(* CoDeSys 2.3 export: PACKML_STATEMODEL_20191003.EXP *)

(* Data type *)
TYPE E_Mode :
(*UserModes: Modes for different production states*)
(
	eMode_undefined := 0,
	eMode_Automatic :=1,
	eMode_Manual :=3,
	eMode_Production1 :=5,
	eMode_Production2 :=6
);
END_TYPE

(* Data type *)
TYPE E_ModeProc :
(*Procedural control modes. Can be changed in any state*)
(
	eModeProc_undefined := 0,
	eModeProc_Automatic :=1,
	eModeProc_SemiAutomatic :=2,
	eModeProc_Manual :=3
);
END_TYPE

(* Data type *)
TYPE E_PackMLState :
(*PackML States*)
(
	eSt_Aborting :=0,
	eSt_Aborted,
	eSt_Clearing,
	eSt_Stopped,
	eSt_Stopping,
	eSt_Resetting,
	eSt_Idle,
	eSt_Starting,
	eSt_Execute,
	eSt_Suspending,
	eSt_Suspended,
	eSt_Unsuspending,
	eSt_Holding,
	eSt_Held,
	eSt_UnHolding,
	eSt_Completing,
	eSt_Completed
);
END_TYPE

(* POU Examples/PRG_MAIN_SAMPLE, ST *)
PROGRAM PRG_MAIN_SAMPLE
VAR
(*	fbStateModel		: FB_PackMLStateModel_ST;	(*FB for executing PackML state model*)		*)
	bBlink				: BOOL;	(*1s blinkg for CodeSys Simulation*)
	c					: INT;	(*Support variable for blinking*)
END_VAR
(* ****** Section 1: Initialisations and default values. Initial conditions for variables on every PLC cycle*)
fbStateModel.bSC := FALSE;

(* ****** Section 2: Grouping PackML states for calling Programs or FB instances.
This is to avoid repetition inside case structure in Section 4. With IF clause setting lower (and upper) state limits we can filter out the states when we 
want to call specific programs. The order of states is defined in Tab:Data types > E_PackMLState. eSt_Aborting is the lowest and eSt_Completed is 
the highest. Here we filter out calling of the programs - we call them only when we are in higher states than Stopped. Inside IF there is again CASE 
which process each Control Mode separately.*)
(*Execution part. Making calls for program if we are on states above Stopped*)
IF (fbStateModel.eState > eSt_Stopped) THEN
	CASE fbStateModel.eMode OF
		(*MODE: MANUAL*)
		eMode_Manual:
			;
		(*MODE: AUTOMATIC*)
		eMode_Automatic:
			;
	END_CASE;
END_IF;

(* ****** Section 3: Actions in your program without considering the Control Mode. I.e. actions are performed same way indenpendent on
current Control Mode selection.*)
(*Mode independent state actions*)
CASE fbStateModel.eState OF
eSt_Aborting:
	(* One can make specific actions in case of specific Mode-State combination.
	   One can also consider to call a specific program when in specific Mode-State combination*)
	actAborting;
	fbStateModel.bSC := TRUE;		(*TODO: Remove/Replace this row with desired actions*)
eSt_Clearing:
	fbStateModel.bSC := TRUE;		(*TODO: Remove/Replace this row with desired actions*)
eSt_Stopping:
	fbStateModel.bSC := TRUE;		(*TODO: Remove/Replace this row with desired actions*)
eSt_Resetting:
	fbStateModel.bSC := TRUE;		(*TODO: Remove/Replace this row with desired actions*)
eSt_Holding:
	fbStateModel.bSC := TRUE;		(*TODO: Remove/Replace this row with desired actions*)
eSt_UnHolding:
	fbStateModel.bSC := TRUE;		(*TODO: Remove/Replace this row with desired actions*)
eSt_Suspending:
	fbStateModel.bSC := TRUE;		(*TODO: Remove/Replace this row with desired actions*)
eSt_Unsuspending:
	fbStateModel.bSC := TRUE;		(*TODO: Remove/Replace this row with desired actions*)
END_CASE;

(* ****** Section 4: Actions in your program which are Control Mode specific. Two nested case structures where outer one selects the
control mode and inner the PackML state. In order to avoid conflicts, it would be better to process each PackML state either in Section 3 
or Section 4, but not in both. *)
(*Execution mode related state actions*)
CASE fbStateModel.eMode OF
(*MODE: MANUAL*)
eMode_Manual:
	(* ****** Section 4.1: PackML state based processing actions when Control Mode is Manual.*)
	CASE fbStateModel.eState OF
	eSt_Idle:
		fbStateModel.bAck_Completed := FALSE;		(*TODO: Remove/Replace this row with desired actions*)
	eSt_Starting:
		fbStateModel.bSC := TRUE;					(*TODO: Remove/Replace this row with desired actions*)
	eSt_Completing:
		fbStateModel.bSC := TRUE;					(*TODO: Remove/Replace this row with desired actions*)
	eSt_Completed:
		fbStateModel.bAck_Completed := TRUE;		(*TODO: Remove/Replace this row with desired actions*)
	END_CASE;

(*MODE: AUTOMATIC*)
eMode_Automatic:
	(* ****** Section 4.2: PackML state based processing actions when Control Mode is Automatic.*)
	CASE fbStateModel.eState OF
	eSt_Idle:
		fbStateModel.bAck_Completed := FALSE;		(*TODO: Remove/Replace this row with desired actions*)
	eSt_Starting:
		fbStateModel.bSC := TRUE;					(*TODO: Remove/Replace this row with desired actions*)
	eSt_Completing:
		fbStateModel.bSC := TRUE;					(*TODO: Remove/Replace this row with desired actions*)
	eSt_Completed:
		;
		(*fbStateModel.bAck_Completed:= TRUE;*)
	END_CASE;

(*MODE: UNKNOWN*)
ELSE	(*This is an Error branch.*)
	; (*TODO: Make implementation*)
END_CASE;

(* ****** Section 5: Calling the fbStateModel instance.
Here the instance of state model is called and all triggering inputs are set, but bSC (State Completed), which you control in your programs. 
This is indication that your program has  finished certain stage.
- Pay attention where the instance fbStateModel is defined. Do you do it in global variables or e.g. here in PRG_MAIN? Important is to use the 
same instance in all places, so that machine state is unique and shared. Remember, if you have multiple definitions, the PRG_MAIN "hides" 
the global one, and might lead to problems elswhere, when you think you are using the same instance, but actually are not. 
- In case you are using the PackML visualisation (VC_PackMLStates), make sure you connect its placeholder to the very same PackML FB instance.
- The Mask for wIgnoreState is created as following. I use binary base for the value(2#). The lowest bit in the mask corresponds the eSt_Aborting
 in E_PackMLState. The next is eSt_Aborted, and so on. Specific state is ignored and jumped over when it is masked out i.e. ignored by having 1 
in that position. Note that implementation allows this only for selected states. See FB_PackMLStateModel_ST code for further details.*)
(*Calling & Updating the state model*)
(*TODO: Evaluate and change all input conditions according your application needs*)
fbStateModel(
	bResetFB:= ,
	eModeReq:= ,
	wIgnoreState := 2#000000,		(*TODO: Which states should be ignodered. Default: 2#000000 or 2#100000*)
	bSC:= ,		(*Must NOT be assigned ANY variable, because fb input is directly assigned above by your programs!!!*)
	bAbort:= ,
	bClear:= ,
	bReset:= ,
	bStart:= ,
	bHold:= ,
	bUn_Hold:= ,
	bSuspend:= ,
	bUn_Suspend:= ,
	bStop:= ,
	bComplete:= ,
	bAck_Completed:= ,
	eMode=> ,
	eState=> );

(* ****** Section 6: Here we update all outputs according the current state of our PackML model. This allows us to process the in single location.
The control of outputs is bind to state, not e.g. to inputs. The inputs are the one driving the PackML model forward. Again CASE structure can be used.*)
(*Call for HMI and UI update*)
HMI_and_UI_Update;
END_PROGRAM
ACTION actAborting:
(*You can add here Aborting related actions as one central collection.
This action can be called from multiple places, in case needed, 
but is part of program*)
;
END_ACTION
ACTION HMI_and_UI_Update:
(*HMI Update*)
(*Calling blinking sub-program*)
(*PRG_Blinking (bSign4Hz=> , bSign2Hz=> , bSign1Hz=> , bSign0_5Hz=> );*)
(*Codesys simulation 1Hz blinking*)
c:= c + 1;
IF c > 1 THEN
	c:=0;
END_IF;
bBlink := (c=0);	(*bBlink is true if c=0*)

(*Init values*)
O_Light_Stop := FALSE;	(*TODO: Change initial values according your app needs*)

(*TODO: Change values according range of states *)
(*Start light*)
(*O_Light_Start :=  (fbStateModel.eState >= eSt_Resetting) AND (fbStateModel.eState < eSt_Completed); *)

(*TODO: Change output values according states *)
CASE fbStateModel.eState OF
eSt_Aborting, eSt_Aborted:
	O_Light_Stop := bBlink;					(*TODO: Change initial values according your app needs*)
eSt_Clearing:
	O_Light_Stop := bBlink; 					(*TODO: Change initial values according your app needs*)
eSt_Stopping, eSt_Stopped, eSt_Completed:
	O_Light_Stop := TRUE;					(*TODO: Change initial values according your app needs*)
eSt_Starting:
	;
	(*O_Light_Start := bBlink;	*)				(*TODO: Change initial values according your app needs*)
END_CASE;
END_ACTION

(* POU Programs/PRG_Blinking, ST *)
PROGRAM PRG_Blinking
(*Avustavia laskentaoperaatioita
- vilkutussignaalit
Author: Niko Siltala, niko.siltala@tut.fi, Tampere University of Technology / MEI
Date: 2016-12-12
Version: 1.0
*)
VAR_OUTPUT
	bSign4Hz:BOOL;					(*4 Hz (240krt/min) taajudella vaihteleva signaali*)
	bSign2Hz:BOOL;					(*2 Hz (120krt/min) taajudella vaihteleva signaali*)
	bSign1Hz:BOOL;					(*1 Hz (60krt/min) taajudella vaihteleva signaali*)
	bSign0_5Hz:BOOL;				(*0,5 Hz (30krt/min) taajudella vaihteleva signaali*)
END_VAR
VAR
	bInitDone	: BOOL	:=FALSE;	(*Ohjelman initialisointi*)
	TP_Delay:TP;				(*Nopein taajuus / 2 tuottaja*)
	bBaseHz:BOOL:=FALSE;		(*Nopein taajuus/2*)
	iBaseHz:UINT:=4;				(*Base taajuus (Hz)*)
	(*RTRIG_BASE: R_TRIG;		(*Base signaali nousee*)*)
	RTRIG_2Hz_Sign : R_TRIG;		(*2Hz signaalin generointi*)
	RTRIG_1Hz_Sign : R_TRIG;		(*1Hz signaalin generointi*)
	RTRIG_0_5Hz_Sign : R_TRIG;	(*0,5Hz signaalin generointi*)
	tBaseTaajuus:TIME;			(*Base vilkutuksen timerin arvo. f/2*)
	fPLC_CYCLE_TIME: LREAL;	(*PLC:n cycli aika. Sekunttia*)

END_VAR
(*Ohjelman initialisoinnit - Suoritetaan vain kertaalleen*)
IF NOT bInitDone THEN
	(*fPLC_CYCLE_TIME := UDINT_TO_LREAL(SystemTaskInfoArr[1].cycleTime) / 10E6; (*[s]*)*)
	fPLC_Cycle_Time := 1;	(*[s]*)
	(*Base Vilkkusignaalien tuottaminen*)
	(* 250ms - 1* cykliaika(20ms)*)
	tBaseTaajuus := LREAL_TO_TIME( ( (1/ UINT_TO_LREAL(iBaseHz) / 2 ) - 1 * fPLC_CYCLE_TIME ) * 1000);
	bInitDone := TRUE;
END_IF;

(*Base signaalin genrointi*)
TP_Delay(IN:=NOT TP_Delay.Q , PT:=tBaseTaajuus);
IF NOT TP_Delay.Q THEN
	bBaseHz := NOT bBaseHz;
	bSign4Hz:= bBaseHz;
END_IF;

(*2Hz signaalin genrointi*)
RTRIG_2Hz_Sign(CLK:=bSign4Hz);
IF RTRIG_2Hz_Sign.Q THEN
	bSign2Hz:=NOT bSign2Hz;
END_IF;

(*1Hz signaalin genrointi*)
RTRIG_1Hz_Sign(CLK:=bSign2Hz);
IF RTRIG_1Hz_Sign.Q THEN
	bSign1Hz:=NOT bSign1Hz;
END_IF;

(*0,5 Hz signaalin generointi*)
RTRIG_0_5Hz_Sign(CLK:=bSign1Hz);
IF (RTRIG_0_5Hz_Sign.Q) THEN
	bSign0_5Hz:= NOT bSign0_5Hz;
END_IF;
END_PROGRAM

(* POU Examples/FB_SFC_Example, SFC *)
FUNCTION_BLOCK FB_SFC_Example
VAR_INPUT
	bReset		: BOOL;	(*Reset Request*)
END_VAR
VAR_OUTPUT
END_VAR
VAR
	bLocalReset	: BOOL;	(*Performs local reset*)
	SFCReset 	: BOOL;	(*Resets the execution of SFC to init once this SFCFlag is set true *)
END_VAR
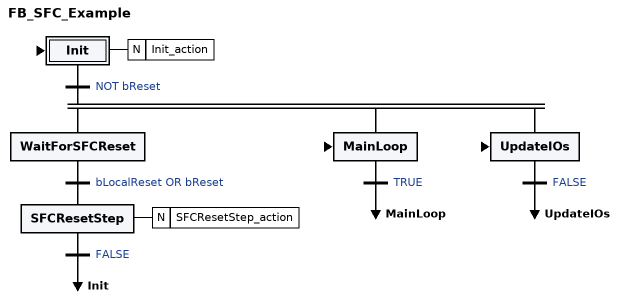
INITIAL_STEP Init:
	Init_action(N);
END_STEP
TRANSITION FROM Init TO (WaitForSFCReset, MainLoop, UpdateIOs) := NOT bReset;
END_TRANSITION
STEP WaitForSFCReset:
END_STEP
TRANSITION FROM WaitForSFCReset TO SFCResetStep := bLocalReset OR bReset;
END_TRANSITION
STEP MainLoop:
END_STEP
TRANSITION FROM MainLoop TO MainLoop := TRUE;
END_TRANSITION
STEP UpdateIOs:
END_STEP
TRANSITION FROM UpdateIOs TO UpdateIOs := FALSE;
END_TRANSITION
STEP SFCResetStep:
	SFCResetStep_action(N);
END_STEP
TRANSITION FROM SFCResetStep TO Init := FALSE;
END_TRANSITION

ACTION Init_action:
SFCReset := FALSE;
bLocalReset	:= FALSE;
END_ACTION

ACTION SFCResetStep_action:
SFCReset := TRUE;
END_ACTION
END_FUNCTION_BLOCK

(* POU FBs/FB_PackMLStateModel_ST, ST *)
FUNCTION_BLOCK FB_PackMLStateModel_ST
(*PackML State model implementation for applications.
Author: Niko Siltala, niko.siltala@tut.fi, Tampere University of Technology / MEI
Date: 2016-12-12
Version: 1.0
*)
VAR_INPUT
	bResetFB	: BOOL;		(*Resets whole FB*)
	eModeReq	: E_Mode;	(*Requested mode*)
	wIgnoreState: DWORD;	(*Ignoring states. See bit from E_PackMLState definition. Aborting = bit0*)
	bSC			: BOOL;		(*Step Completed acknoledgement*)
	bAbort		: BOOL;		(*Abortting signal = EmergencyStop*)
	bClear		: BOOL;		(*Clear signal*)
	bReset		: BOOL;		(*Reseting signal*)
	bStart		: BOOL;		(*Start signal*)
	bHold		: BOOL;		(*Hold signal*)
	bUn_Hold	: BOOL;		(*Un-Hold signal*)
	bSuspend	: BOOL;		(*Suspend signal*)
	bUn_Suspend	: BOOL;		(*Un-Suspend signal*)
	bStop		: BOOL;		(*Stop signal*)
	bComplete	: BOOL;		(*Complete signal*)
	bAck_Completed	: BOOL;	(*Acknoledgement for Complete signal*)
END_VAR
VAR_OUTPUT
	eMode	: E_Mode;		(*Current mode*)
	eState	: E_PackMLState;(*Current state*)
	strState : STRING(15);		(*State as String*)
END_VAR
VAR
	RTrig_bSC		: R_TRIG; 		(*Rising trigger for State Completed*)
	RTrig_StateChange : R_TRIG; 	(*Rising trigger for State signal*)
	bResetLocal		: BOOL:=FALSE;	(*Paikallinen Reset*)
	bInitDone		: BOOL;			(*Initialisation*)
END_VAR
IF bResetFB THEN	(*Reseting FB*)
	bInitDone := FALSE;
END_IF;

(*Initialisation*)
IF NOT bInitDone THEN
	eState:= eSt_Aborting;
	strState:='Aborting';
	bInitDone:=TRUE;
END_IF;

(*Rising triggers monitor*)
RTrig_bSC(CLK:=bSC , Q=> );

(*Abort signal interrupt*)
IF bAbort AND (eState > eSt_Clearing) THEN
	eState:=eSt_Aborting;
END_IF;

(*Stop signal interrupt*)
IF bStop AND (eState > eSt_Stopping) THEN
	eState:=eSt_Stopping;
END_IF;


(*Main case structure*)
CASE eState OF
eSt_Aborting:
	strState:='Aborting';
	IF bSC THEN
		eState:=eSt_Aborted;
	END_IF;

eSt_Aborted:
	strState:='Aborted';
	eMode:=eModeReq;	(*Change Mode allowed*)
	IF bClear AND NOT bAbort THEN
		eState:=eSt_Clearing;
	END_IF;

eSt_Clearing:
	strState:='Clearing';
	IF bAbort THEN
		eState:=eSt_Aborting;
	ELSIF bSC THEN
		eState:=eSt_Stopped;
		RTrig_StateChange(CLK:=bReset , Q=> );
	END_IF;

eSt_Stopping:
	strState:='Stopping';
	IF bSC THEN
		eState:=eSt_Stopped;
		RTrig_StateChange(CLK:=bReset , Q=> );
	END_IF;

eSt_Stopped:
	strState:='Stopped';
	eMode:=eModeReq;	(*Change Mode allowed*)
	RTrig_StateChange(CLK:=bReset , Q=> );
(*	ELSIF NOT bStop AND (RTrig_StateChange.Q OR (wIgnoreState.5 AND bStart) ) THEN*)
	IF NOT bStop THEN	(*Stop signal is not active.*)
		IF wIgnoreState.5 AND bStart THEN	(*Reset state is ignored and going directly to start *)
			eState:=eSt_Idle;
(*		ELSIF RTrig_StateChange.Q THEN 	(*Rising edge for reset*)*)
		ELSIF bReset THEN 	(*Reset*)
			eState:=eSt_Resetting;
		END_IF;
	END_IF;

eSt_Resetting:
	strState:='Resetting';
	IF bSC OR wIgnoreState.5 THEN
		eState:=eSt_Idle;
	END_IF;

eSt_Idle:
	strState:='Idle';
	eMode:=eModeReq;	(*Change Mode allowed*)
	IF bStart OR wIgnoreState.6 THEN (* IDLE state is ignoered*)
		eState:=eSt_Starting;
	END_IF;

eSt_Starting:
	strState:='Starting';
	IF bSC OR wIgnoreState.7 THEN (* STARTING state is ignoered*)
		eState:=eSt_Execute;
	END_IF;

eSt_Execute:
	strState:='Execute';
	IF bComplete THEN
		eState:=eSt_Completing;
	ELSIF bHold THEN
		eState:=eSt_Holding;
	ELSIF bSuspend THEN
		eState:=eSt_Suspending;
	END_IF;

eSt_Holding:
	strState:='Holding';
	IF bSC THEN
		eState:=eSt_Held;
	END_IF;

eSt_Held:
	strState:='Held';
	IF bUn_Hold AND NOT bHold THEN
		eState:=eSt_UnHolding;
	END_IF;

eSt_UnHolding:
	strState:='Un-Holding';
	IF bSC THEN
		eState:=eSt_Execute;
	END_IF;

eSt_Suspending:
	strState:='Suspending';
	IF bSC THEN
		eState:=eSt_Suspended;
	END_IF;

eSt_Suspended:
	strState:='Suspended';
	IF bUn_Suspend AND NOT bSuspend THEN
		eState:=eSt_Unsuspending;
	END_IF;

eSt_Unsuspending:
	strState:='Un-Suspending';
	IF bSC THEN
		eState:=eSt_Execute;
	END_IF;

eSt_Completing:
	strState:='Completing';
	IF RTrig_bSC.Q THEN
		eState:=eSt_Completed;
	END_IF;

eSt_Completed:
	strState:='Completed';
	IF bReset OR bAck_Completed THEN
		eState:=eSt_Resetting;
	END_IF;

ELSE
	(*Default error handler. Undefined state set*)
	eState:=eSt_Aborting;
END_CASE;
END_FUNCTION_BLOCK

(* Visualisation VC_PackMLStates
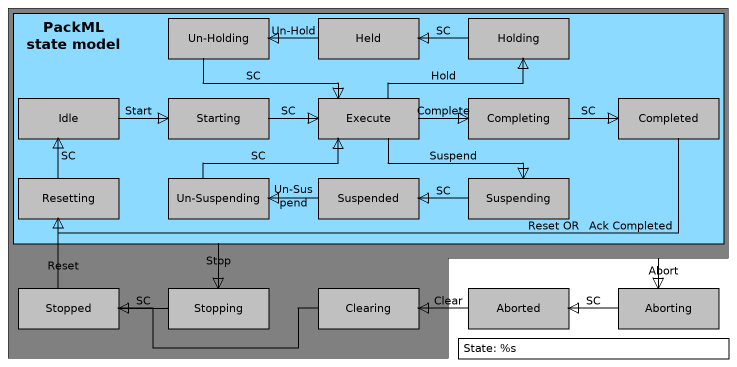
rounded rectangle at (160,280)-(261,321): text "Stopping"; alarm colour if $PackML$.eState = 4
rounded rectangle at (10,90)-(111,131): text "Idle"; alarm colour if $PackML$.eState = 6
rounded rectangle at (160,170)-(261,211): text "Un-Suspending"; alarm colour if $PackML$.eState = 11
rounded rectangle at (610,280)-(711,321): text "Aborting"; alarm colour if $PackML$.eState = 0
rounded rectangle at (460,280)-(561,321): text "Aborted"; alarm colour if $PackML$.eState = 1
rectangle at (450,330)-(721,351): text "State: %s"; shows $PackML$.strState
rounded rectangle at (310,280)-(411,321): text "Clearing"; alarm colour if $PackML$.eState = 2
rounded rectangle at (10,280)-(111,321): text "Stopped"; alarm colour if $PackML$.eState = 3
rounded rectangle at (10,170)-(111,211): text "Resetting"; alarm colour if $PackML$.eState = 5
rounded rectangle at (160,90)-(261,131): text "Starting"; alarm colour if $PackML$.eState = 7
rounded rectangle at (310,90)-(411,131): text "Execute"; alarm colour if $PackML$.eState = 8
rounded rectangle at (460,90)-(561,131): text "Completing"; alarm colour if $PackML$.eState = 15
rounded rectangle at (610,90)-(711,131): text "Completed"; alarm colour if $PackML$.eState = 16
rounded rectangle at (310,170)-(411,211): text "Suspended"; alarm colour if $PackML$.eState = 10
rounded rectangle at (460,170)-(561,211): text "Suspending"; alarm colour if $PackML$.eState = 9
rounded rectangle at (460,10)-(561,51): text "Holding"; alarm colour if $PackML$.eState = 12
rounded rectangle at (310,10)-(411,51): text "Held"; alarm colour if $PackML$.eState = 13
rounded rectangle at (160,10)-(261,51): text "Un-Holding"; alarm colour if $PackML$.eState = 14
polyline at (645,250)-(655,280): alarm colour if $PackML$.bAbort
rectangle at (635,255)-(676,271): text "Abort"; alarm colour if $PackML$.bAbort
polyline at (205,235)-(215,280): alarm colour if $PackML$.bStop
rectangle at (190,245)-(231,261): text "Stop"; alarm colour if $PackML$.bStop
polyline at (195,130)-(335,170): alarm colour if $PackML$.bSC
rectangle at (235,140)-(266,156): text "SC"; alarm colour if $PackML$.bSC
polyline at (195,50)-(335,90): alarm colour if $PackML$.bSC
polyline at (380,50)-(520,90): alarm colour if $PackML$.bHold
rectangle at (420,60)-(451,76): text "Hold"; alarm colour if $PackML$.bHold
polyline at (560,295)-(610,305): alarm colour if $PackML$.bSC
polyline at (45,210)-(55,280): alarm colour if $PackML$.bReset
polyline at (110,105)-(160,115): alarm colour if $PackML$.bStart
polyline at (110,295)-(310,340): alarm colour if $PackML$.bSC
rectangle at (230,60)-(261,76): text "SC"; alarm colour if $PackML$.bSC
polyline at (380,130)-(520,170): alarm colour if $PackML$.bSuspend
rectangle at (415,140)-(476,156): text "Suspend"; alarm colour if $PackML$.bSuspend
rectangle at (120,285)-(151,301): text "SC"; alarm colour if $PackML$.bSC
rectangle at (570,285)-(601,301): text "SC"; alarm colour if $PackML$.bSC
polyline at (410,295)-(460,305): alarm colour if $PackML$.bClear
rectangle at (420,285)-(461,301): text "Clear"; alarm colour if $PackML$.bClear
polyline at (260,105)-(310,115): alarm colour if $PackML$.bSC
rectangle at (265,95)-(296,111): text "SC"; alarm colour if $PackML$.bSC
rectangle at (110,95)-(151,111): text "Start"; alarm colour if $PackML$.bStart
rectangle at (35,250)-(76,266): text "Reset"; alarm colour if $PackML$.bReset
polyline at (410,185)-(460,195): alarm colour if $PackML$.bSC
rectangle at (420,175)-(451,191): text "SC"; alarm colour if $PackML$.bSC
polyline at (410,25)-(460,35): alarm colour if $PackML$.bSC
rectangle at (420,15)-(451,31): text "SC"; alarm colour if $PackML$.bSC
polyline at (260,185)-(310,195): alarm colour if $PackML$.bUn_Suspend
rectangle at (260,170)-(311,206): text "Un-Sus / pend"; alarm colour if $PackML$.bUn_Suspend
polyline at (260,25)-(310,35): alarm colour if $PackML$.bUn_Hold
rectangle at (260,15)-(311,31): text "Un-Hold"; alarm colour if $PackML$.bUn_Hold
polyline at (410,105)-(460,115): alarm colour if $PackML$.bComplete
rectangle at (410,95)-(461,111): text "Complete"; alarm colour if $PackML$.bComplete
polyline at (560,105)-(610,115): alarm colour if $PackML$.bSC
rectangle at (565,95)-(596,111): text "SC"; alarm colour if $PackML$.bSC
polyline at (45,130)-(55,170): alarm colour if $PackML$.bSC
rectangle at (45,140)-(76,156): text "SC"; alarm colour if $PackML$.bSC
polyline at (50,130)-(670,225): alarm colour if $PackML$.bReset OR $PackML$.Ack_Completed
rectangle at (515,210)-(576,226): text "Reset OR"; alarm colour if $PackML$.bReset
rectangle at (575,210)-(671,226): text "Ack Completed"; alarm colour if $PackML$.bAck_Completed
rectangle at (10,10)-(121,51): text "PackML / state model"
2 more shapes without text or variables
*)
